(* Logix 5000 project; controller START_STOP Emulate 5570 rev 30.12; software revision 30.00 *)

TASK MainTask (continuous, watchdog 500 ms) : MainProgram

MODULES
   Local : Emulate 5570 (ICP 2, rev 30.12)
      VIRTUAL_OUTPUTS : vendor 1 type 0 code 15 (ICP 4, rev 1.1, Output RPI 50 ms)
      VIRTUAL_INPUTS : vendor 1 type 0 code 15 (ICP 3, rev 1.1, Output RPI 50 ms)
END_MODULES

VAR_GLOBAL   (* controller tags *)
   CVY_8 : ALIAS FOR Local:4:O.Data[0].3;
   CVY_8_DN : BOOL;
   DEL_1 : TIMER := (PRE := 1000);
   DEL_2 : TIMER := (PRE := 1000);
   FIN_SP1 : ALIAS FOR Local:3:I.Data[1].2;
   FIN_SP2 : ALIAS FOR Local:3:I.Data[1].3;
   PB_CVY_8 : ALIAS FOR Local:3:I.Data[1].4;
   PRUEBA : BOOL;
   SP1_DN : BOOL;
   SP2_DN : BOOL;
   SR1 : BOOL;
   SR2 : BOOL;
   Started : ALIAS FOR Local:4:O.Data[0].0;
   STP_g : ALIAS FOR Local:3:I.Data[1].1;
   STT_g : ALIAS FOR Local:3:I.Data[1].0;
   STT_SP1 : ALIAS FOR Local:4:O.Data[0].1;
   STT_SP2 : ALIAS FOR Local:4:O.Data[0].2;
END_VAR

PROGRAM MainProgram   (* main routine MainRoutine *)

ROUTINE Encendido_CVY8   (* ladder *)
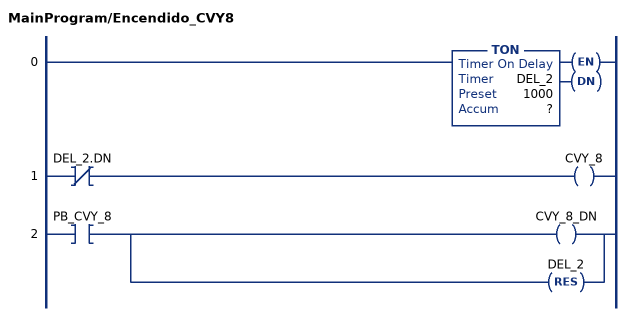
   0: TON(DEL_2,?,?);
   1: XIO(DEL_2.DN)OTE(CVY_8);
   2: XIC(PB_CVY_8)[OTE(CVY_8_DN) ,RES(DEL_2) ];
END_ROUTINE

ROUTINE Inicio_Soplado   (* ladder *)
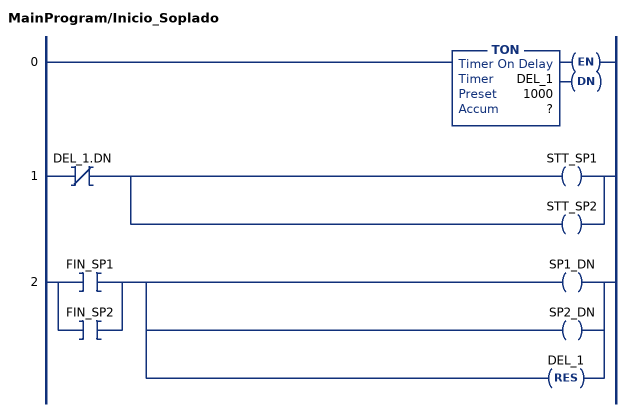
   0: TON(DEL_1,?,?);
   1: XIO(DEL_1.DN)[OTE(STT_SP1) ,OTE(STT_SP2) ];
   2: [XIC(FIN_SP1) ,XIC(FIN_SP2) ][OTE(SP1_DN) ,OTE(SP2_DN) ,RES(DEL_1) ];
END_ROUTINE

ROUTINE MainRoutine   (* ladder *)
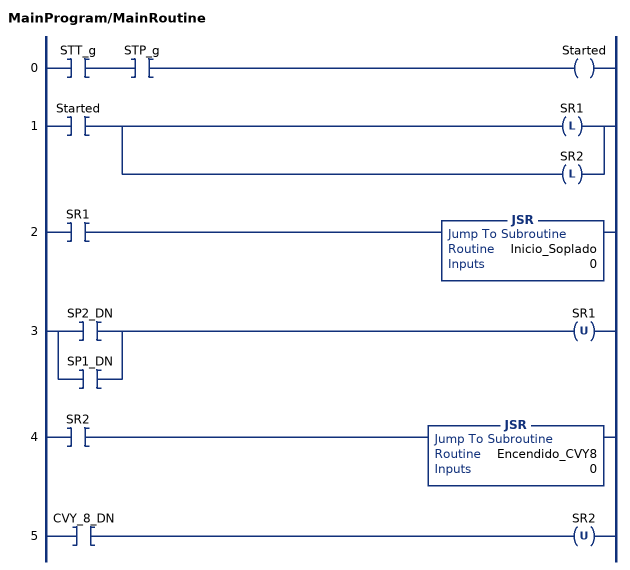
   0: XIC(STT_g)XIC(STP_g)OTE(Started);
   1: XIC(Started)[OTL(SR1) ,OTL(SR2) ];
   2: XIC(SR1)JSR(Inicio_Soplado,0);
   3: [XIC(SP2_DN) ,XIC(SP1_DN) ]OTU(SR1);
   4: XIC(SR2)JSR(Encendido_CVY8,0);
   5: XIC(CVY_8_DN)OTU(SR2);
END_ROUTINE
END_PROGRAM
